{attribute 'linkalways'} 
{attribute 'no_explicit_call' := 'This FB is a CLASS and must be accessed using methods or properties'}
{attribute 'enable_dynamic_creation'}
FUNCTION_BLOCK _ETcVnOcrOptions EXTENDS EnumDatatypeBase
VAR
	localData : ETcVnOcrOptions;
	activeData : REFERENCE TO ETcVnOcrOptions;
	enumBaseDatatype : _UDINT(localData);
END_VAR

METHOD PRIVATE AddLocalEnumeration
VAR_INPUT
	Enumeration : T_MAXSTRING;
	Value : ETcVnOcrOptions;
END_VAR
AddEnumeration(Enumeration, Value);
END_METHOD

PROPERTY PUBLIC Address : PVOID
GET
Address := ADR(activeData);
END_GET
END_PROPERTY

METHOD PUBLIC ClearReference
VAR_INPUT
END_VAR
activeData REF= localData;
SetBaseDatatypeReference();
END_METHOD

METHOD PUBLIC Clone : I_Datatype
VAR
    pClone : POINTER TO _ETcVnOcrOptions;
END_VAR
pClone := __NEW(_ETcVnOcrOptions(InitialValue := Value));
Clone := pClone^;
END_METHOD

METHOD FB_init : BOOL
VAR_INPUT
	bInitRetains : BOOL; // if TRUE, the retain variables are initialized (warm start / cold start)
	bInCopyCode : BOOL;  // if TRUE, the instance afterwards gets moved into the copy code (online change)
	InitialValue : ETcVnOcrOptions;
END_VAR
localData := InitialValue;
AddBaseDatatype(enumBaseDatatype);
ClearReference();

AddLocalEnumeration('TCVN_OO_WITHBLANKS', ETcVnOcrOptions.TCVN_OO_WITHBLANKS);
END_METHOD

PROPERTY PUBLIC Identifier : T_MAXSTRING
GET
Identifier := 'ETcVnOcrOptions';
END_GET
END_PROPERTY

METHOD IsEnumeratorValueEqual : BOOL
VAR_INPUT
	Enumerator : I_KeyValueForwardEnumerator;
END_VAR
VAR
	storedValue : ETcVnOcrOptions;
END_VAR
IF NOT Enumerator.TryGet(storedValue) THEN
	RETURN;
END_IF

IsEnumeratorValueEqual := storedValue = activeData;
END_METHOD

METHOD PUBLIC MakeReferenceTo
VAR_INPUT
	ReferenceTarget : REFERENCE TO ETcVnOcrOptions;
END_VAR
activeData REF= ReferenceTarget;
SetBaseDatatypeReference();
END_METHOD

METHOD PROTECTED SetBaseDatatypeReference
VAR_INPUT
END_VAR
enumBaseDatatype.MakeReferenceTo(activeData);
END_METHOD

PROPERTY PUBLIC Size : UDINT
GET
Size := SIZEOF(activeData);
END_GET
END_PROPERTY

METHOD TryMakeReferenceTo : BOOL
VAR_INPUT
	Target : I_Datatype;
END_VAR
VAR
	targetAsEnum : I_EnumDatatype;
	pTargetData : POINTER TO ETcVnOcrOptions;
END_VAR
IF NOT Target.TryResolveAsEnumDatatype(targetAsEnum) THEN
	RETURN;
END_IF

IF targetAsEnum.Identifier <> Identifier THEN
	RETURN;
END_IF

pTargetData := Target.Address;
activeData REF= pTargetData^;
SetBaseDatatypeReference();
TryMakeReferenceTo := TRUE;
END_METHOD

PROPERTY PUBLIC Value : ETcVnOcrOptions
GET
Value := activeData;
END_GET
SET
activeData := Value;
END_SET
END_PROPERTY

END_FUNCTION_BLOCK

(* stored: Version 1.1.0.1, ProductVersion 3.1.4024.13
   POU _ETcVnOcrOptions: Id {c29854d3-3fca-0fbf-3a61-47df1e1f8d67}, SpecialFunc None
   Folder Core: Id {5ff367a7-847b-0eb8-1fa2-38822f4dcef6}
   Folder Protected: Id {a1787d22-0259-0b14-237d-7690055da0f4}
   Folder Customize: Id {ad891574-9ad6-00cd-33ac-476f0b75d049}
   Folder Constructor: Id {6f846874-f96f-0768-3ba6-e35c49f6d7b1}
   Folder Private: Id {42d577a5-7d9e-0056-05da-79461a381c0b}
   Folder Protected: Id {5f56281e-11f7-0a72-2803-addf801ae45e}
   Method AddLocalEnumeration: Id {b8709ce2-3a51-09b4-3e38-45964587dde0}
   Property Address: Id {8fa8cbcc-dc8a-01b2-0a9e-7129fd4bd4b2}
   Get Get: Id {c2d6f0da-bd27-0ad2-14f1-5a25a3b7e216}
   Method ClearReference: Id {b4844477-4161-0d63-02cf-9d29cf8470bc}
   Method Clone: Id {d99d5e16-4c6e-030a-33bd-8dc745342c75}
   Method FB_init: Id {8c3b47b6-b07d-09b8-0861-610f2bd648e9}
   Property Identifier: Id {5f307b6f-38fe-03fd-3523-e6026d9eead8}
   Get Get: Id {055dd11c-d996-046f-2b54-2e0ecf183207}
   Method IsEnumeratorValueEqual: Id {6c03672d-462c-0852-279c-6e497aebbcc4}
   Method MakeReferenceTo: Id {aa8a3b29-f877-0b2a-092d-2d0af7bd234e}
   Method SetBaseDatatypeReference: Id {a9e60ab4-6798-04b6-275b-466c554580ee}
   Property Size: Id {493f2e8c-6e26-0674-111f-403945a14fe6}
   Get Get: Id {1c5cb55c-2369-071d-171a-03faa8ff36be}
   Method TryMakeReferenceTo: Id {55be9424-529e-04f6-1d05-0eb2f52de9c3}
   Property Value: Id {42f1b535-ceb2-0066-2d0c-6d8e7334d2a1}
   Get Get: Id {2256db4d-9e25-0a6c-0b9a-f94f6e9154a6}
   Set Set: Id {a8dd7c52-0e4c-085d-2181-9f7fc9daa638} *)
